// TIA Portal V19 export
TYPE "C402_STU_AFS_IF_VKL_TYPIC"
   STRUCT
      CMD_HND { ExternalAccessible := 'False'; ExternalVisible := 'False'; ExternalWritable := 'False'} : Bool;   // Commando Bedieningsmode Hand activeren
      CMD_HND_ROOD { ExternalAccessible := 'False'; ExternalVisible := 'False'; ExternalWritable := 'False'} : Bool;   // Handmatig commando Rood
      CMD_HND_GROE { ExternalAccessible := 'False'; ExternalVisible := 'False'; ExternalWritable := 'False'} : Bool;   // Handmatig commando Groen
      CMD_HND_KNIP { ExternalAccessible := 'False'; ExternalVisible := 'False'; ExternalWritable := 'False'} : Bool;   // Handmatig commando Geel Knipperen
      CMD_HND_UIT { ExternalAccessible := 'False'; ExternalVisible := 'False'; ExternalWritable := 'False'} : Bool;   // Handmatig commando Uit
      STO_ROOD { ExternalAccessible := 'False'; ExternalVisible := 'False'; ExternalWritable := 'False'} : Bool;   // Geen enkel verkeerslicht kan de stand rood tonen
   END_STRUCT;
END_TYPE
